{attribute 'qualified_only'}
VAR_GLOBAL
	uDcvEnableMainJib : BOOL := TRUE;		//Enable/Disable manual control of MainJibCylinder valve
	uDcvMainJib : LREAL;
	uDcvEnableKnuckleJib : BOOL := TRUE;			//Enable/Disable manual control of BoomCylinder valve
	uDcvKnuckleJib : LREAL;
END_VAR

(* stored: Version 1.1.0.1, ProductVersion 3.1.4024.9
   GVL Inputs: Id {379b0098-5f22-4bf9-b1bd-8bcf308b02e1} *)
